(* PLC project PROGRAM_13_12_OPC, Phoenix Contact PC WORX 6.30 *)
(* stored: companyURL www.kw-software.com, creationDateTime 2016-01-09T01:01:39, version 1452297699, modificationDateTime 2016-01-09T01:01:39 *)

FUNCTION_BLOCK Przyklad

						
							
						
					
END_FUNCTION_BLOCK
